// SIMATIC S7-200 project (STEP 7-Micro/WIN), CPU 224XP CN REL 02.01

ORGANIZATION_BLOCK MAIN:OB1
TITLE=
BEGIN
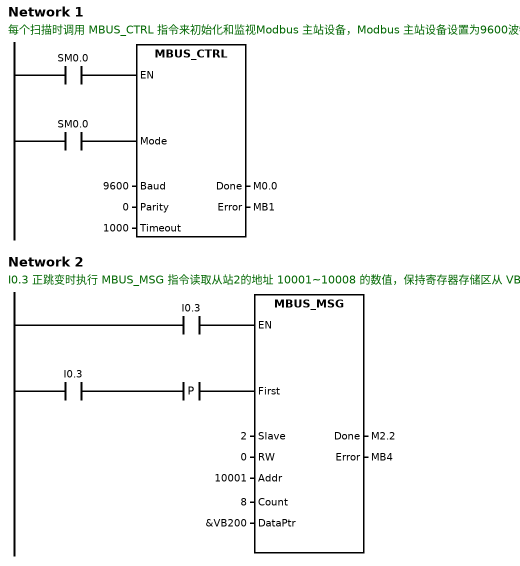
Network 1
// 每个扫描时调用 MBUS_CTRL 指令来初始化和监视Modbus 主站设备，Modbus 主站设备设置为9600波特率，无奇偶校验，允许从站1000毫秒(1秒)的应答时间
// (network saved uncompiled; LAD cells follow)
// row 0: c0 -| |- SM0.0  c1 [MBUS_CTRL EN:=power@row0, Mode:=power@row1, Baud:=9600, Parity:=0, Timeout:=1000, Done=>M0.0, Error=>MB1]
// row 1: c0 -| |- SM0.0  c1 [box]
// row 2: c1 [box]
Network 2
// I0.3 正跳变时执行 MBUS_MSG 指令读取从站2的地址 10001~10008 的数值，保持寄存器存储区从 VB200 开始，长8个字。根据 Modbus 从站寻址方法，10001~10008 即 S7-200 PLC 中I0.1~I0.7的 Modbus 地址值
// (network saved uncompiled; LAD cells follow)
// row 0: c0 --  c1 -| |- I0.3  c2 [MBUS_MSG EN:=power@row0, First:=power@row1, Slave:=2, RW:=0, Addr:=10001, Count:=8, DataPtr:=&VB200, Done=>M2.2, Error=>MB4]
// row 1: c0 -| |- I0.3  c1 -|P|-  c2 [box]
// row 2: c2 [box]
// row 3: c2 [box]
END_ORGANIZATION_BLOCK

// SBR1: protected block, not included

// SBR2: protected block, not included

// SBR3: protected block, not included

// SBR4: protected block, not included

// SBR5: protected block, not included

// SBR6: protected block, not included
